{attribute 'qualified_only'}
{attribute 'strict'}
TYPE StateVe :
(
	Off,
	Fill,
	Idle,
	Eject,
	Done,
	Error
);
END_TYPE

(* stored: Version 1.1.0.1, ProductVersion 3.1.4024.3
   DUT StateVe: Id {42c2aca7-6a3a-46cb-b3fc-d0d17b24100b} *)
